
TYPE "TimeTest_001"
STRUCT
        SIMPLE_SECOND : TIME;
        MILLISECONDS : TIME;
        HOUR_AND_HALF : TIME;
        COMPLEX_TIME : TIME;
        TWO_DAYS : TIME;
        TIME_ARRAY : ARRAY[0..5] OF TIME;
        EQUIVALENT_TIMES : ARRAY[0..2] OF TIME;
        COMPLEX_TIME_ARRAY : ARRAY[0..2] OF TIME;
END_STRUCT;
END_TYPE